// TIA Portal V20 export
DATA_BLOCK "IDB_BarcodeReader"   // DB29
// stored: InstanceOfName ProductionLine.BarcodeReader, InstanceOfType FB, Namespace ProductionLine
"ProductionLine.BarcodeReader"
   // VAR
   //    DP1 : "Global.DataMan262";
   //    DP2 : "Global.DataMan262";
   //    DP3 : "Global.DataMan262";
   //    DP4 : "Global.DataMan262";
   // END_VAR
BEGIN
END_DATA_BLOCK
